RoboDK station: main.rdk

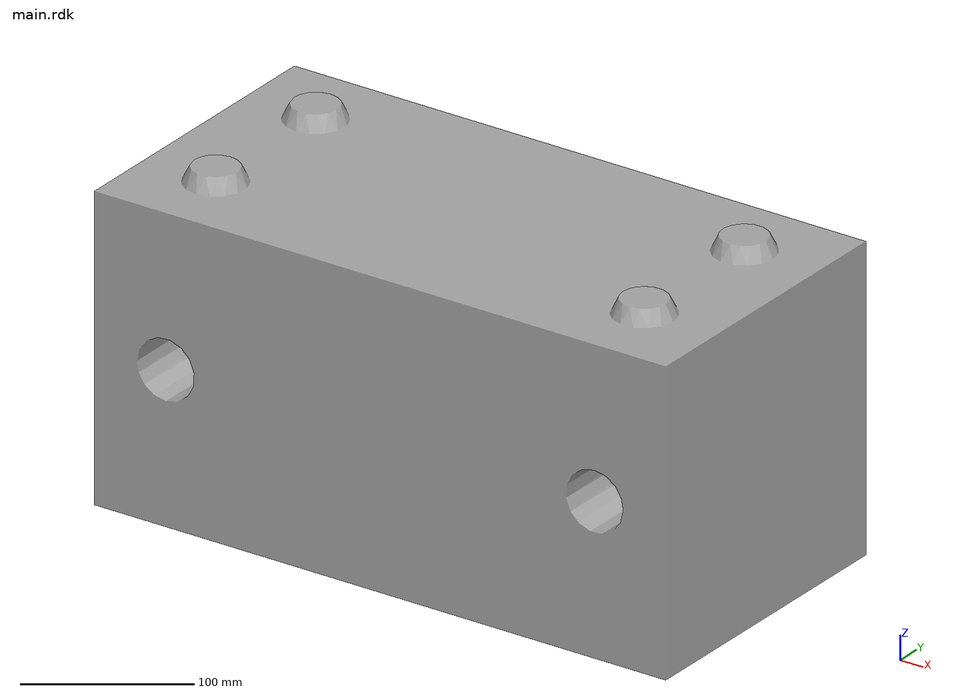
[picture v0: the station drawn from its stored meshes, robots at their saved joint values, targets as dots, program paths as lines]
Station main (saved by RoboDK 5.4.1). Poses are relative to the parent item; angles as X-Y-Z fixed-axis rotations.
  - object brick at (0, 0, 0) mm, size 400 x 200 x 210 mm, geometry from brick.stp
